{attribute 'pack_mode' := '1'}
TYPE ST_Enable EXTENDS ST_PLCMsg:
STRUCT
END_STRUCT
END_TYPE

(* stored: Version 1.1.0.1, ProductVersion 3.1.4022.18
   DUT ST_Enable: Id {215e77ac-23bf-47b6-b5dd-027108da9b7d} *)
